    movel([0.332496, -1.166919, -2.692890, -0.852580, 1.570796, 1.903292],accel_mss,speed_ms,0,blend_radius_m)
    movel([0.332398, -1.167537, -2.692618, -0.852234, 1.570796, 1.903194],accel_mss,speed_ms,0,blend_radius_m)
    movel([0.332125, -1.167972, -2.692426, -0.851991, 1.570796, 1.902922],accel_mss,speed_ms,0,blend_radius_m)
    movel([0.331713, -1.168242, -2.692306, -0.851841, 1.570796, 1.902510],accel_mss,speed_ms,0,blend_radius_m)
    movel([0.331306, -1.168113, -2.692363, -0.851912, 1.570796, 1.902103],accel_mss,speed_ms,0,blend_radius_m)
    movel([0.331181, -1.167790, -2.692506, -0.852093, 1.570796, 1.901977],accel_mss,speed_ms,0,blend_radius_m)
    movel([0.330747, -1.166094, -2.693253, -0.853042, 1.570796, 1.901543],accel_mss,speed_ms,0,blend_radius_m)
    speed_ms = 0.005
    movel([0.330747, -1.156321, -2.688286, -0.867781, 1.570796, 1.901543],accel_mss,speed_ms,0,blend_radius_m)
    speed_ms = 0.040
    movel([0.331469, -1.169115, -2.682650, -0.860624, 1.570796, 1.902266],accel_mss,speed_ms,0,blend_radius_m)
    speed_ms = 0.005
    movel([0.331469, -1.178854, -2.687559, -0.845975, 1.570796, 1.902266],accel_mss,speed_ms,0,blend_radius_m)
    speed_ms = 0.025
    movel([0.330682, -1.179241, -2.687384, -0.845764, 1.570796, 1.901478],accel_mss,speed_ms,0,blend_radius_m)
    movel([0.330527, -1.179246, -2.687382, -0.845761, 1.570796, 1.901324],accel_mss,speed_ms,0,blend_radius_m)
    movel([0.330285, -1.179088, -2.687453, -0.845847, 1.570796, 1.901081],accel_mss,speed_ms,0,blend_radius_m)
    movel([0.330236, -1.178791, -2.687588, -0.846010, 1.570796, 1.901032],accel_mss,speed_ms,0,blend_radius_m)
    movel([0.330383, -1.178440, -2.687747, -0.846202, 1.570796, 1.901179],accel_mss,speed_ms,0,blend_radius_m)
    movel([0.330690, -1.178117, -2.687893, -0.846379, 1.570796, 1.901487],accel_mss,speed_ms,0,blend_radius_m)
    movel([0.331117, -1.177631, -2.688113, -0.846646, 1.570796, 1.901914],accel_mss,speed_ms,0,blend_radius_m)
    movel([0.331243, -1.177291, -2.688266, -0.846832, 1.570796, 1.902040],accel_mss,speed_ms,0,blend_radius_m)
    movel([0.331366, -1.176749, -2.688511, -0.847130, 1.570796, 1.902162],accel_mss,speed_ms,0,blend_radius_m)
    movel([0.331570, -1.174446, -2.689546, -0.848397, 1.570796, 1.902366],accel_mss,speed_ms,0,blend_radius_m)
    movel([0.331243, -1.172459, -2.690434, -0.849496, 1.570796, 1.902040],accel_mss,speed_ms,0,blend_radius_m)
    movel([0.330392, -1.170834, -2.691158, -0.850397, 1.570796, 1.901188],accel_mss,speed_ms,0,blend_radius_m)
    movel([0.329032, -1.169616, -2.691698, -0.851074, 1.570796, 1.899828],accel_mss,speed_ms,0,blend_radius_m)
    movel([0.328083, -1.169161, -2.691900, -0.851328, 1.570796, 1.898879],accel_mss,speed_ms,0,blend_radius_m)
    movel([0.325708, -1.168715, -2.692097, -0.851577, 1.570796, 1.896504],accel_mss,speed_ms,0,blend_radius_m)
    movel([0.324679, -1.168798, -2.692061, -0.851531, 1.570796, 1.895475],accel_mss,speed_ms,0,blend_radius_m)
    movel([0.323933, -1.169040, -2.691953, -0.851395, 1.570796, 1.894730],accel_mss,speed_ms,0,blend_radius_m)
    movel([0.323752, -1.169240, -2.691865, -0.851284, 1.570796, 1.894548],accel_mss,speed_ms,0,blend_radius_m)
    movel([0.323250, -1.170060, -2.691501, -0.850827, 1.570796, 1.894046],accel_mss,speed_ms,0,blend_radius_m)
    movel([0.322821, -1.170309, -2.691391, -0.850689, 1.570796, 1.893618],accel_mss,speed_ms,0,blend_radius_m)
    movel([0.322188, -1.170348, -2.691374, -0.850667, 1.570796, 1.892984],accel_mss,speed_ms,0,blend_radius_m)
    movel([0.321130, -1.170170, -2.691453, -0.850767, 1.570796, 1.891926],accel_mss,speed_ms,0,blend_radius_m)
    movel([0.319263, -1.170120, -2.691475, -0.850794, 1.570796, 1.890059],accel_mss,speed_ms,0,blend_radius_m)
    movel([0.318553, -1.170236, -2.691423, -0.850729, 1.570796, 1.889350],accel_mss,speed_ms,0,blend_radius_m)
    movel([0.316685, -1.170740, -2.691199, -0.850449, 1.570796, 1.887481],accel_mss,speed_ms,0,blend_radius_m)
    movel([0.315326, -1.171430, -2.690893, -0.850066, 1.570796, 1.886122],accel_mss,speed_ms,0,blend_radius_m)
    movel([0.314393, -1.172331, -2.690491, -0.849566, 1.570796, 1.885189],accel_mss,speed_ms,0,blend_radius_m)
    movel([0.313800, -1.173463, -2.689986, -0.848940, 1.570796, 1.884596],accel_mss,speed_ms,0,blend_radius_m)
    movel([0.313494, -1.174437, -2.689549, -0.848402, 1.570796, 1.884291],accel_mss,speed_ms,0,blend_radius_m)
    movel([0.312668, -1.174607, -2.689473, -0.848309, 1.570796, 1.883464],accel_mss,speed_ms,0,blend_radius_m)
    movel([0.311909, -1.174837, -2.689370, -0.848182, 1.570796, 1.882705],accel_mss,speed_ms,0,blend_radius_m)
    movel([0.311134, -1.175217, -2.689200, -0.847972, 1.570796, 1.881930],accel_mss,speed_ms,0,blend_radius_m)
    movel([0.309598, -1.176378, -2.688677, -0.847333, 1.570796, 1.880394],accel_mss,speed_ms,0,blend_radius_m)
    movel([0.308951, -1.177067, -2.688367, -0.846955, 1.570796, 1.879747],accel_mss,speed_ms,0,blend_radius_m)
    movel([0.308397, -1.177815, -2.688030, -0.846545, 1.570796, 1.879194],accel_mss,speed_ms,0,blend_radius_m)
    movel([0.308016, -1.178523, -2.687709, -0.846157, 1.570796, 1.878812],accel_mss,speed_ms,0,blend_radius_m)
    movel([0.307480, -1.180072, -2.687007, -0.845310, 1.570796, 1.878276],accel_mss,speed_ms,0,blend_radius_m)
    movel([0.307253, -1.180364, -2.686874, -0.845151, 1.570796, 1.878050],accel_mss,speed_ms,0,blend_radius_m)
    movel([0.306952, -1.180575, -2.686778, -0.845036, 1.570796, 1.877749],accel_mss,speed_ms,0,blend_radius_m)
    movel([0.306688, -1.180630, -2.686754, -0.845006, 1.570796, 1.877485],accel_mss,speed_ms,0,blend_radius_m)
    movel([0.306514, -1.180523, -2.686802, -0.845064, 1.570796, 1.877310],accel_mss,speed_ms,0,blend_radius_m)
    movel([0.306409, -1.179886, -2.687092, -0.845412, 1.570796, 1.877206],accel_mss,speed_ms,0,blend_radius_m)
    movel([0.306585, -1.179075, -2.687459, -0.845855, 1.570796, 1.877381],accel_mss,speed_ms,0,blend_radius_m)
    movel([0.306955, -1.178226, -2.687844, -0.846319, 1.570796, 1.877751],accel_mss,speed_ms,0,blend_radius_m)
    movel([0.307530, -1.177295, -2.688264, -0.846830, 1.570796, 1.878326],accel_mss,speed_ms,0,blend_radius_m)
    movel([0.308227, -1.176405, -2.688665, -0.847318, 1.570796, 1.879023],accel_mss,speed_ms,0,blend_radius_m)
    movel([0.309047, -1.175553, -2.689049, -0.847787, 1.570796, 1.879843],accel_mss,speed_ms,0,blend_radius_m)
    movel([0.309945, -1.174793, -2.689390, -0.848206, 1.570796, 1.880741],accel_mss,speed_ms,0,blend_radius_m)
    movel([0.310844, -1.174197, -2.689657, -0.848535, 1.570796, 1.881640],accel_mss,speed_ms,0,blend_radius_m)
    movel([0.311760, -1.173751, -2.689857, -0.848781, 1.570796, 1.882556],accel_mss,speed_ms,0,blend_radius_m)
    movel([0.312381, -1.173381, -2.690023, -0.848986, 1.570796, 1.883177],accel_mss,speed_ms,0,blend_radius_m)
    movel([0.312612, -1.173117, -2.690140, -0.849131, 1.570796, 1.883408],accel_mss,speed_ms,0,blend_radius_m)
    movel([0.313295, -1.172066, -2.690609, -0.849713, 1.570796, 1.884092],accel_mss,speed_ms,0,blend_radius_m)
    movel([0.313953, -1.171357, -2.690925, -0.850107, 1.570796, 1.884749],accel_mss,speed_ms,0,blend_radius_m)
    movel([0.315643, -1.170069, -2.691497, -0.850822, 1.570796, 1.886439],accel_mss,speed_ms,0,blend_radius_m)
    movel([0.316858, -1.169488, -2.691755, -0.851146, 1.570796, 1.887654],accel_mss,speed_ms,0,blend_radius_m)
    movel([0.318433, -1.169018, -2.691963, -0.851408, 1.570796, 1.889230],accel_mss,speed_ms,0,blend_radius_m)
    movel([0.320036, -1.168735, -2.692088, -0.851566, 1.570796, 1.890833],accel_mss,speed_ms,0,blend_radius_m)
    movel([0.322567, -1.168740, -2.692086, -0.851563, 1.570796, 1.893364],accel_mss,speed_ms,0,blend_radius_m)
    movel([0.322872, -1.168592, -2.692151, -0.851645, 1.570796, 1.893669],accel_mss,speed_ms,0,blend_radius_m)
    movel([0.324135, -1.167670, -2.692559, -0.852160, 1.570796, 1.894931],accel_mss,speed_ms,0,blend_radius_m)
    movel([0.324975, -1.167402, -2.692677, -0.852310, 1.570796, 1.895771],accel_mss,speed_ms,0,blend_radius_m)
    movel([0.327374, -1.167417, -2.692670, -0.852301, 1.570796, 1.898171],accel_mss,speed_ms,0,blend_radius_m)
    movel([0.328614, -1.167684, -2.692553, -0.852152, 1.570796, 1.899410],accel_mss,speed_ms,0,blend_radius_m)
    movel([0.329739, -1.168112, -2.692364, -0.851913, 1.570796, 1.900535],accel_mss,speed_ms,0,blend_radius_m)
    movel([0.330655, -1.168678, -2.692114, -0.851597, 1.570796, 1.901451],accel_mss,speed_ms,0,blend_radius_m)
    movel([0.331414, -1.169411, -2.691789, -0.851189, 1.570796, 1.902210],accel_mss,speed_ms,0,blend_radius_m)
    movel([0.332359, -1.171022, -2.691074, -0.850293, 1.570796, 1.903155],accel_mss,speed_ms,0,blend_radius_m)
    movel([0.332853, -1.172983, -2.690200, -0.849206, 1.570796, 1.903649],accel_mss,speed_ms,0,blend_radius_m)
    movel([0.332875, -1.175166, -2.689222, -0.848000, 1.570796, 1.903671],accel_mss,speed_ms,0,blend_radius_m)
    movel([0.332415, -1.177444, -2.688197, -0.846748, 1.570796, 1.903211],accel_mss,speed_ms,0,blend_radius_m)
    movel([0.332236, -1.177958, -2.687965, -0.846466, 1.570796, 1.903033],accel_mss,speed_ms,0,blend_radius_m)
    movel([0.331821, -1.178571, -2.687687, -0.846130, 1.570796, 1.902617],accel_mss,speed_ms,0,blend_radius_m)
    movel([0.331469, -1.178854, -2.687559, -0.845975, 1.570796, 1.902266],accel_mss,speed_ms,0,blend_radius_m)
    movel([0.330682, -1.179241, -2.687384, -0.845764, 1.570796, 1.901478],accel_mss,speed_ms,0,blend_radius_m)
    movel([0.330527, -1.179246, -2.687382, -0.845761, 1.570796, 1.901324],accel_mss,speed_ms,0,blend_radius_m)
    movel([0.330285, -1.179088, -2.687453, -0.845847, 1.570796, 1.901081],accel_mss,speed_ms,0,blend_radius_m)
    movel([0.330236, -1.178791, -2.687588, -0.846010, 1.570796, 1.901032],accel_mss,speed_ms,0,blend_radius_m)
    movel([0.330383, -1.178440, -2.687747, -0.846202, 1.570796, 1.901179],accel_mss,speed_ms,0,blend_radius_m)
    movel([0.330690, -1.178117, -2.687893, -0.846379, 1.570796, 1.901487],accel_mss,speed_ms,0,blend_radius_m)
    movel([0.331117, -1.177631, -2.688113, -0.846646, 1.570796, 1.901914],accel_mss,speed_ms,0,blend_radius_m)
    movel([0.331194, -1.177425, -2.688206, -0.846759, 1.570796, 1.901990],accel_mss,speed_ms,0,blend_radius_m)
    speed_ms = 0.005
    movel([0.331194, -1.167681, -2.683290, -0.861418, 1.570796, 1.901990],accel_mss,speed_ms,0,blend_radius_m)
    speed_ms = 0.040
    movel([0.330295, -1.185364, -2.675246, -0.851779, 1.570796, 1.901092],accel_mss,speed_ms,0,blend_radius_m)
    speed_ms = 0.005
    movel([0.330295, -1.195055, -2.680082, -0.837252, 1.570796, 1.901092],accel_mss,speed_ms,0,blend_radius_m)
    speed_ms = 0.025
    movel([0.330668, -1.194304, -2.680435, -0.837650, 1.570796, 1.901464],accel_mss,speed_ms,0,blend_radius_m)
    movel([0.331756, -1.190620, -2.682157, -0.839612, 1.570796, 1.902552],accel_mss,speed_ms,0,blend_radius_m)
    movel([0.332001, -1.189344, -2.682750, -0.840295, 1.570796, 1.902797],accel_mss,speed_ms,0,blend_radius_m)
    movel([0.332119, -1.187217, -2.683735, -0.841437, 1.570796, 1.902916],accel_mss,speed_ms,0,blend_radius_m)
    movel([0.331930, -1.185198, -2.684665, -0.842526, 1.570796, 1.902726],accel_mss,speed_ms,0,blend_radius_m)
    movel([0.331458, -1.183462, -2.685461, -0.843466, 1.570796, 1.902255],accel_mss,speed_ms,0,blend_radius_m)
    movel([0.330731, -1.182191, -2.686042, -0.844156, 1.570796, 1.901527],accel_mss,speed_ms,0,blend_radius_m)
    movel([0.329629, -1.181311, -2.686443, -0.844634, 1.570796, 1.900425],accel_mss,speed_ms,0,blend_radius_m)
    movel([0.328223, -1.180944, -2.686610, -0.844834, 1.570796, 1.899019],accel_mss,speed_ms,0,blend_radius_m)
    movel([0.326708, -1.181131, -2.686525, -0.844733, 1.570796, 1.897505],accel_mss,speed_ms,0,blend_radius_m)
    movel([0.325994, -1.181415, -2.686396, -0.844578, 1.570796, 1.896790],accel_mss,speed_ms,0,blend_radius_m)
    movel([0.325287, -1.181850, -2.686198, -0.844341, 1.570796, 1.896083],accel_mss,speed_ms,0,blend_radius_m)
    movel([0.324302, -1.182566, -2.685871, -0.843952, 1.570796, 1.895099],accel_mss,speed_ms,0,blend_radius_m)
    movel([0.323465, -1.182020, -2.686120, -0.844249, 1.570796, 1.894261],accel_mss,speed_ms,0,blend_radius_m)
    movel([0.322422, -1.181476, -2.686368, -0.844545, 1.570796, 1.893218],accel_mss,speed_ms,0,blend_radius_m)
    movel([0.321330, -1.181177, -2.686505, -0.844708, 1.570796, 1.892126],accel_mss,speed_ms,0,blend_radius_m)
    movel([0.320125, -1.181111, -2.686534, -0.844743, 1.570796, 1.890921],accel_mss,speed_ms,0,blend_radius_m)
    movel([0.318743, -1.181273, -2.686461, -0.844655, 1.570796, 1.889539],accel_mss,speed_ms,0,blend_radius_m)
    movel([0.317778, -1.181473, -2.686370, -0.844546, 1.570796, 1.888574],accel_mss,speed_ms,0,blend_radius_m)
    movel([0.316559, -1.181932, -2.686160, -0.844297, 1.570796, 1.887355],accel_mss,speed_ms,0,blend_radius_m)
    movel([0.315884, -1.182337, -2.685976, -0.844077, 1.570796, 1.886681],accel_mss,speed_ms,0,blend_radius_m)
    movel([0.314583, -1.183372, -2.685502, -0.843515, 1.570796, 1.885380],accel_mss,speed_ms,0,blend_radius_m)
    movel([0.313518, -1.184598, -2.684940, -0.842850, 1.570796, 1.884314],accel_mss,speed_ms,0,blend_radius_m)
    movel([0.313020, -1.185597, -2.684481, -0.842310, 1.570796, 1.883816],accel_mss,speed_ms,0,blend_radius_m)
    movel([0.313023, -1.185910, -2.684337, -0.842142, 1.570796, 1.883819],accel_mss,speed_ms,0,blend_radius_m)
    movel([0.313225, -1.186073, -2.684262, -0.842054, 1.570796, 1.884022],accel_mss,speed_ms,0,blend_radius_m)
    movel([0.313519, -1.186017, -2.684288, -0.842084, 1.570796, 1.884316],accel_mss,speed_ms,0,blend_radius_m)
    movel([0.313889, -1.185759, -2.684407, -0.842223, 1.570796, 1.884685],accel_mss,speed_ms,0,blend_radius_m)
    movel([0.314227, -1.185384, -2.684579, -0.842425, 1.570796, 1.885023],accel_mss,speed_ms,0,blend_radius_m)
    movel([0.314428, -1.184999, -2.684756, -0.842633, 1.570796, 1.885224],accel_mss,speed_ms,0,blend_radius_m)
    movel([0.314724, -1.184554, -2.684961, -0.842874, 1.570796, 1.885520],accel_mss,speed_ms,0,blend_radius_m)
    movel([0.315577, -1.183834, -2.685291, -0.843264, 1.570796, 1.886373],accel_mss,speed_ms,0,blend_radius_m)
    movel([0.316521, -1.183156, -2.685601, -0.843632, 1.570796, 1.887317],accel_mss,speed_ms,0,blend_radius_m)
    movel([0.317247, -1.182786, -2.685771, -0.843833, 1.570796, 1.888043],accel_mss,speed_ms,0,blend_radius_m)
    movel([0.318828, -1.182430, -2.685933, -0.844026, 1.570796, 1.889624],accel_mss,speed_ms,0,blend_radius_m)
    movel([0.320459, -1.182511, -2.685896, -0.843982, 1.570796, 1.891256],accel_mss,speed_ms,0,blend_radius_m)
    movel([0.321949, -1.182993, -2.685676, -0.843720, 1.570796, 1.892745],accel_mss,speed_ms,0,blend_radius_m)
    movel([0.323647, -1.184304, -2.685075, -0.843009, 1.570796, 1.894444],accel_mss,speed_ms,0,blend_radius_m)
    movel([0.324065, -1.184366, -2.685047, -0.842976, 1.570796, 1.894861],accel_mss,speed_ms,0,blend_radius_m)
    movel([0.324491, -1.184104, -2.685167, -0.843118, 1.570796, 1.895287],accel_mss,speed_ms,0,blend_radius_m)
    movel([0.325034, -1.183433, -2.685475, -0.843481, 1.570796, 1.895830],accel_mss,speed_ms,0,blend_radius_m)
    movel([0.325654, -1.182744, -2.685790, -0.843856, 1.570796, 1.896450],accel_mss,speed_ms,0,blend_radius_m)
    movel([0.326005, -1.182575, -2.685867, -0.843947, 1.570796, 1.896801],accel_mss,speed_ms,0,blend_radius_m)
    movel([0.327349, -1.182292, -2.685996, -0.844101, 1.570796, 1.898145],accel_mss,speed_ms,0,blend_radius_m)
    movel([0.328009, -1.182344, -2.685972, -0.844072, 1.570796, 1.898806],accel_mss,speed_ms,0,blend_radius_m)
    movel([0.329157, -1.182899, -2.685719, -0.843771, 1.570796, 1.899953],accel_mss,speed_ms,0,blend_radius_m)
    movel([0.330016, -1.184055, -2.685190, -0.843144, 1.570796, 1.900813],accel_mss,speed_ms,0,blend_radius_m)
    movel([0.330553, -1.185780, -2.684397, -0.842212, 1.570796, 1.901349],accel_mss,speed_ms,0,blend_radius_m)
    movel([0.330759, -1.187424, -2.683639, -0.841326, 1.570796, 1.901555],accel_mss,speed_ms,0,blend_radius_m)
    movel([0.330735, -1.188977, -2.682920, -0.840492, 1.570796, 1.901531],accel_mss,speed_ms,0,blend_radius_m)
    movel([0.330462, -1.190688, -2.682125, -0.839576, 1.570796, 1.901258],accel_mss,speed_ms,0,blend_radius_m)
    movel([0.329269, -1.195207, -2.680010, -0.837172, 1.570796, 1.900065],accel_mss,speed_ms,0,blend_radius_m)
    movel([0.329333, -1.195452, -2.679895, -0.837042, 1.570796, 1.900129],accel_mss,speed_ms,0,blend_radius_m)
    movel([0.329574, -1.195507, -2.679869, -0.837013, 1.570796, 1.900370],accel_mss,speed_ms,0,blend_radius_m)
    movel([0.329774, -1.195449, -2.679897, -0.837044, 1.570796, 1.900571],accel_mss,speed_ms,0,blend_radius_m)
    movel([0.330295, -1.195055, -2.680082, -0.837252, 1.570796, 1.901092],accel_mss,speed_ms,0,blend_radius_m)
    movel([0.330668, -1.194304, -2.680435, -0.837650, 1.570796, 1.901464],accel_mss,speed_ms,0,blend_radius_m)
    movel([0.331348, -1.191998, -2.681514, -0.838876, 1.570796, 1.902144],accel_mss,speed_ms,0,blend_radius_m)
    speed_ms = 0.005
    movel([0.331348, -1.145970, -2.656733, -0.909686, 1.570796, 1.902144],accel_mss,speed_ms,0,blend_radius_m)
    speed_ms = 1.000
    movel([0.331348, -1.145970, -2.656733, -0.909686, 1.570796, 1.902144],accel_mss,speed_ms,0,blend_radius_m)
    # Splitting Linear movement in 6 (instruction 8476: MoveL 8167)
    movel([0.331348, -1.112111, -2.635138, -0.965140, 1.570796, 1.902144],accel_mss,speed_ms,0,blend_radius_m)
    movel([0.331348, -1.082005, -2.612778, -1.017606, 1.570796, 1.902144],accel_mss,speed_ms,0,blend_radius_m)
    movel([0.331348, -1.055344, -2.589727, -1.067318, 1.570796, 1.902144],accel_mss,speed_ms,0,blend_radius_m)
    movel([0.331348, -1.031836, -2.566048, -1.114505, 1.570796, 1.902144],accel_mss,speed_ms,0,blend_radius_m)
    movel([0.331348, -1.011208, -2.541797, -1.159385, 1.570796, 1.902144],accel_mss,speed_ms,0,blend_radius_m)
    movel([0.331348, -0.993207, -2.517018, -1.202164, 1.570796, 1.902144],accel_mss,speed_ms,0,blend_radius_m)
    # End of main program
  end

  Machining1()
end
